PROGRAM MAIN
VAR
END_VAR

Auto_Manual();
Emergency_Stop();

END_PROGRAM

(* stored: Version 1.1.0.1, ProductVersion 3.1.4024.12
   POU MAIN: Id {54befd21-3517-4010-bc97-4f29dd46757e}, SpecialFunc None *)
